METHOD PRIVATE stageEx : BOOL
VAR_IN_OUT
	robot : RobotA21;
	aoiTemplate : AOI_StagingTemplate;
	aoiStaging : AOI_StageWoodBunk;
	stageStep : INT;
END_VAR
VAR_INPUT
	includeTop, includeLeft, includeRight, includeBottom : BOOL;
END_VAR
VAR_OUTPUT
	error : BOOL;
END_VAR
{warning disable C0371}
IF robot.error THEN
	error := TRUE;
	RETURN;
ELSIF robot.reservation <> sectionID AND_THEN NOT robot.reserve(sectionID) THEN
	RETURN;
ELSIF robot.tool <> sectionID AND_THEN NOT robot.changeEOAT(targetTool := sectionID) THEN
	RETURN;
END_IF

CASE stageStep OF
	0: //generate staging template
		IF aoiTemplate.done THEN
			aoiTemplate.execute := FALSE;
			stageStep := 10;
			RETURN;
		END_IF
		
		aoiTemplate.execute := NOT aoiTemplate.busy;
		
		aoiTemplate.includeTop := includeTop;
		aoiTemplate.includeLeft := includeLeft;
		aoiTemplate.includeRight := includeRight;
		aoiTemplate.includeBottom := includeBottom;
		
	10: //stage tables
		IF aoiStaging.slot > 10 THEN
			aoiStaging.execute := FALSE;			
			stageStep := COMPLETE;
			RETURN;
		END_IF
		
		aoiStaging.execute := NOT aoiStaging.busy; //execute if aoiStaging is ready
		
		aoiStaging.slot := MAX(1, aoiStaging.slot); //if 0, sets to 1
		aoiStaging.slot := MIN(aoiStaging.slot, 999); //prevents overflow 
		
		IF aoiStaging.donePulse THEN
			aoiStaging.slot := aoiStaging.slot + 1;
		END_IF
	
	COMPLETE:
		aoiTemplate.clearTemplate();
		aoiTemplate.execute := FALSE;
		aoiStaging.execute := FALSE;
		aoiStaging.reset();
		
		robot.release(sectionID);
		
		aoiStaging.slot := 0;
		
		stageEx := TRUE;
		//stageStep := 0;
END_CASE

error := aoiStaging.error;
END_METHOD

METHOD PROTECTED usesProcess : BOOL
VAR
	i : INT;
END_VAR
FOR i:=0 TO GVL.maxPairs BY 1 DO
	IF PositionIsValid(materialsArr[i]) THEN
		usesProcess := TRUE;
		RETURN;
	END_IF
END_FOR
END_METHOD

METHOD PROTECTED validateInsertion : BOOL
VAR_INPUT
	checkTop : BOOL;
	checkLeft : BOOL;
	checkRight : BOOL;
	checkBottom : BOOL;
END_VAR
validateInsertion := 
	(NOT checkTop OR_ELSE SuctionQuality(suctions:= suctionTop)) AND
	(NOT checkLeft OR_ELSE SuctionQuality(suctions:= suctionLeft)) AND
	(NOT checkRight OR_ELSE SuctionQuality(suctions:= suctionRight)) AND
	(NOT checkBottom OR_ELSE SuctionQuality(suctions:= suctionBottom));

(*
validateSuctionQuality := 
	(
		NOT checkTop OR_ELSE InsertionQuality(
			suctions:= suctionTop, 
			insertionMaterial:= loadedMaterials[Surface.TOP], 
			recipeMaterial:= materialsArr[iPair].top)
	) AND
	(
		NOT checkLeft OR_ELSE InsertionQuality(
			suctions:= suctionLeft, 
			insertionMaterial:= loadedMaterials[Surface.LEFT], 
			recipeMaterial:= materialsArr[iPair].left)
	) AND
	(
		NOT checkRight OR_ELSE InsertionQuality(
			suctions:= suctionRight, 
			insertionMaterial:= loadedMaterials[Surface.RIGHT], 
			recipeMaterial:= materialsArr[iPair].right)
	) AND
	(
		NOT checkBottom OR_ELSE InsertionQuality(
			suctions:= suctionBottom, 
			insertionMaterial:= loadedMaterials[Surface.BOTTOM], 
			recipeMaterial:= materialsArr[iPair].bottom)
	);
*)
END_METHOD

END_FUNCTION_BLOCK

// ---- Sections/Abstract/SectionEx.TcPOU
FUNCTION_BLOCK ABSTRACT SectionEx
VAR_INPUT
	enable : BOOL;
	sectionID : SectionEnum;
	
	firstConveyor : INT;
	lastConveyor : INT;
END_VAR
VAR_IN_OUT
	bundlesQueue : ARRAY[*] OF Bundle;
	bundlesBypass : ARRAY[*] OF BOOL; //if true, then bypass current bundle
END_VAR
VAR_OUTPUT
	bundleOut : Bundle; //assigned if there is a bundle to target
	bypass : BOOL; //assigned once the bundle head passes the section (status >= ACTIVE)
END_VAR
VAR_OUTPUT //PackML states + controls
	pmlModeString : STRING;
	pmlStateString : STRING;
	
	stop : BOOL;
	execute : BOOL;
	hold : BOOL;
	reset : BOOL;
	
	ready : BOOL;
	busy : BOOL;
	done : BOOL;
	error : BOOL;
	backlog : BOOL;
	
	iBundle : INT(0..GVL.maxQueue);
	iPair : INT(0..GVL.maxPairs);
END_VAR
VAR
	pmlState : E_PMLState;
	pmlCommand : E_PMLCommand;
	pmlStateMachine : PML_StateMachine;
	
	pmlModeRequest : E_PMLCustomUnitMode := ePMLCustomUnitMode_Production;
	pmlMode : E_PMLCustomUnitMode;
	pmlModeManager : PML_UnitModeManager;
END_VAR
VAR
	currentBundle : REFERENCE TO Bundle;
	currentBypass : REFERENCE TO BOOL;
	
	loaded : BOOL;
	loadedMaterials : ARRAY[Surface.TOP..Surface.BOTTOM_RIGHT] OF STRING;
	
	entryRefPos : (*REFERENCE TO*) REAL;
	exitRefPos : (*REFERENCE TO*) REAL;
	
	requestedConveyorMode : ConveyorMode;
	
	nextSection : POINTER TO SectionEx;
	prevSection : POINTER TO SectionEx;
	
	occupied : BOOL; //may need to move this to Hardware GVL since this is a sensor
	
	status : SectionTask; //section status
END_VAR
VAR_STAT CONSTANT
	INCLUSIVE : INT := 0;
	EXCLUSIVE : INT := 1;
	COMPLETE : INT := 1030;
	
	suctionReleaseDelay : TIME := T#1000MS;
END_VAR

currentBundle REF= bundlesQueue[iBundle];
currentBypass REF= bundlesBypass[iBundle];
bypass := currentBypass;

ready := status = 0;
busy := status > 0;
done := done;
error := error;
backlog := iBundle >= GVL.maxQueue;

callLocalModules();
blocks();

pmlStates();

METHOD assignConveyors : BOOL
VAR_INPUT
	conveyorStart : INT;
	conveyorEnd : INT;
END_VAR
firstConveyor := conveyorStart;
lastConveyor := conveyorEnd;

assignConveyors := TRUE;
END_METHOD

METHOD PROTECTED blocks : BOOL
VAR_INPUT
END_VAR
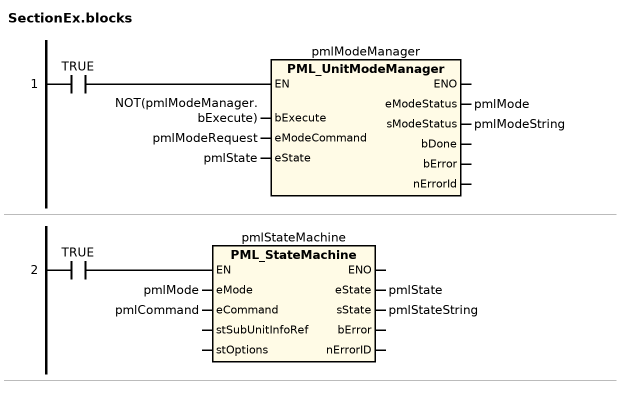
// NETWORK 1
pmlModeManager(
    bExecute := NOT(pmlModeManager.bExecute),
    eModeCommand := pmlModeRequest,
    eState := pmlState,
    eModeStatus => pmlMode,
    sModeStatus => pmlModeString); // PML_UnitModeManager

// NETWORK 2
pmlStateMachine(eMode := pmlMode, eCommand := pmlCommand, eState => pmlState, sState => pmlStateString); // PML_StateMachine
END_METHOD

METHOD PROTECTED ABSTRACT callLocalModules : BOOL
END_METHOD

METHOD connectTo : BOOL
VAR_INPUT
	connectedSection : POINTER TO SectionEx;
END_VAR
nextSection := connectedSection;

IF connectedSection <> 0 THEN
	connectedSection^.prevSection := THIS;
END_IF
END_METHOD

METHOD PROTECTED directionCheckAndSet : BOOL
VAR_INPUT
	conveyorRef : REAL;
	target : REAL;
END_VAR
//returns true conveyorRef is in range of target
IF InRange(conveyorRef - GVL.precisionTolerance, conveyorRef + GVL.precisionTolerance, target, EXCLUSIVE) THEN
	directionCheckAndSet := TRUE;
	
ELSIF conveyorRef > target THEN
	pConveyorMode := ConveyorMode.BACKWARD;
	
ELSIF conveyorRef < target THEN
	pConveyorMode := ConveyorMode.FORWARD;
	
END_IF
END_METHOD

METHOD PROTECTED ABSTRACT discharge : BOOL
VAR_INPUT
END_VAR
(*
unload, unstage, etc
*)
END_METHOD

METHOD PROTECTED ABSTRACT load : BOOL
VAR_INPUT
	pairIndex : INT;
END_VAR
VAR_OUTPUT
	error : BOOL;
END_VAR
(*
loading takes place while the section is NOT active
materials are loaded for the next incoming bundle, not the current bundle - may differ for each section
*)
END_METHOD

METHOD PROTECTED ABSTRACT maintenance : BOOL
VAR_INPUT
END_VAR
END_METHOD

PROPERTY PROTECTED pConveyorMode : ConveyorMode
GET
pConveyorMode := requestedConveyorMode;
END_GET
SET
VAR
	i : DINT;
END_VAR
requestedConveyorMode := pConveyorMode;

FOR i:=firstConveyor TO lastConveyor BY 1 DO
	
	CASE status OF
		SectionTask.ALIGNING, -100:
			//all conveyors requested to same mode
			conveyorsArr[i]^.setRequest(requestedConveyorMode);
			
		SectionTask.ACTIVE, SectionTask.CLEARING:
			//once previous bundle catches up, the conveyor that bundle sits on must be linked to this section
			//a conveyor control module will handle linking
			
			IF conveyorsArr[i]^.IsOccupied THEN //follow this section's request
				conveyorsArr[i]^.setRequest(requestedConveyorMode);
				
			ELSE //catch up succeeding bundle (FOLLOW PREVIOUS SECTION)
				IF prevSection <> 0 THEN
					conveyorsArr[i]^.setRequest( prevSection^.pConveyorMode );
				END_IF
			END_IF
	END_CASE	
	
END_FOR
END_SET
END_PROPERTY

METHOD PROTECTED pmlStates : BOOL
(*
PackML
	state machine for packaging applications - see Tc3_PackML_V2 library on InfoSys
	
	final states - wait for an input or condition and command to new state
	intermediate states - complete a task and call pmlStateMachine.M_StateComplete() to advance to next state
	
the following states currently use the same logic (albeit in different methods), implementation may change later
	ps_Stopping() and ps_Aborting()
	ps_Resetting() and ps_Clearing()
	
STOP - controlled stop **with intent to shutdown or vacate for extended time** induced by operator/HMI - otherwise use HOLD
ABORT - emergency stop due to machine errors


HOLD - minor local issues
SUSPEND - external issues

EXECUTE - major control logic
	different modes may require different tasks
	create methods as required for different modes, then call the correct method in ps_Completing()
	can be commanded to STOP, ABORT, HOLD, or SUSPEND at any point
COMPLETING - process complete, move product out of system and finish transition to COMPLETED

the implementation below can be copied to all POUs that use a PackML state machine
the individual ps_< > methods need to be implemented for the specific application
*)
IF ps_AbortCondition() THEN //abort condition
	pmlCommand := ePMLCommand_Abort;
ELSIF ps_StopCondition() THEN //stop condition
	pmlCommand := ePMLCommand_Stop;
END_IF

CASE pmlState OF
	0 (*ePMLState_Undefined*): //default state on startup
		pmlCommand := ePMLCommand_Stop;
		
	ePMLState_Stopping:
		IF ps_Stopping() THEN
			pmlStateMachine.M_StateComplete();
		END_IF
		
	ePMLState_Stopped:
		IF ps_Stopped() THEN
			pmlCommand := ePMLCommand_Reset;
		END_IF
	
    ePMLState_Resetting:
		IF ps_Resetting() THEN
			pmlStateMachine.M_StateComplete();
		END_IF
		
	ePMLState_Idle:
		IF ps_Idle() THEN
			pmlCommand := ePMLCommand_Start;
		END_IF		
	
	ePMLState_Starting:
		IF ps_Starting() THEN
			pmlStateMachine.M_StateComplete();
		END_IF
	
	ePMLState_Execute: //check the conditions in order of their priority, currently HOLD has the highest priority
		IF ps_HoldCondition() THEN
			pmlCommand := ePMLCommand_Hold;
			
		ELSIF ps_SuspendCondition() THEN
			pmlCommand := ePMLCommand_Suspend;			
		
		ELSIF ps_Execute(error => error) THEN //ps_Execute.error => THIS^.error
			pmlStateMachine.M_StateComplete();
			pmlCommand := ePMLCommand_Complete;
		END_IF
		
	ePMLState_Completing:
		IF ps_Completing() THEN
			pmlStateMachine.M_StateComplete();
		END_IF
	
	ePMLState_Complete:
		IF ps_Complete() THEN
			pmlCommand := ePMLCommand_Reset;
		END_IF
	
	ePMLState_Holding:
		IF ps_Holding() THEN
			pmlStateMachine.M_StateComplete();
		END_IF
	
	ePMLState_Held:
		IF NOT hold THEN
			pmlCommand := ePMLCommand_Unhold;
		END_IF
	
	ePMLState_Unholding:
		IF ps_Unholding() THEN
			pmlStateMachine.M_StateComplete(); //release all pause commands and IO
		END_IF
		
	ePMLState_Suspending: //based on next section conditions
		IF ps_Suspending() THEN
			pmlStateMachine.M_StateComplete();
		END_IF
		
	ePMLState_Suspended: //based on next section conditions
		IF ps_Suspended() THEN
			pmlCommand := ePMLCommand_Unsuspend;
		END_IF
	
	ePMLState_Unsuspending: //based on next section conditions
		IF ps_Unsuspending() THEN
			pmlStateMachine.M_StateComplete();
		END_IF
	
	ePMLState_Aborting:
		IF ps_Aborting() THEN
			pmlStateMachine.M_StateComplete();
		END_IF
	
	ePMLState_Aborted:
		IF ps_Aborted() THEN
			pmlCommand := ePMLCommand_Clear;
		END_IF
	
	ePMLState_Clearing:
		IF ps_Clearing() THEN
			pmlStateMachine.M_StateComplete();
		END_IF
	
END_CASE
END_METHOD

METHOD PROTECTED ABSTRACT process : BOOL
VAR_INPUT
	auto : BOOL;
END_VAR
VAR_OUTPUT
	error : BOOL;
END_VAR
(*
this method is implemented by each section according to their material packaging steps
*)
END_METHOD

METHOD PROTECTED ABSTRACT ps_AbortCondition : BOOL
VAR_INPUT
END_VAR
END_METHOD

METHOD PROTECTED ABSTRACT ps_Aborted : BOOL
VAR_INPUT
END_VAR
END_METHOD

METHOD PROTECTED ABSTRACT ps_Aborting : BOOL
VAR_INPUT
END_VAR
END_METHOD

METHOD PROTECTED ABSTRACT ps_Clearing : BOOL
VAR_INPUT
END_VAR
END_METHOD

METHOD PROTECTED ABSTRACT ps_Complete : BOOL
VAR_INPUT
END_VAR
END_METHOD

METHOD PROTECTED ABSTRACT ps_Completing : BOOL
VAR_INPUT
END_VAR
END_METHOD

METHOD PROTECTED ps_Execute : BOOL
VAR_INPUT
END_VAR
VAR_OUTPUT
	error : BOOL;
END_VAR
CASE pmlMode OF
	0: //invalid mode
	ePMLCustomUnitMode_Production:		ps_Execute := runSectionTasks(auto := TRUE);
	ePMLCustomUnitMode_Maintenance:		maintenance();
	ePMLCustomUnitMode_Manual:			//
	ePMLCustomUnitMode_SemiAuto:		ps_Execute := runSectionTasks(auto := FALSE);
END_CASE
END_METHOD

METHOD PROTECTED ABSTRACT ps_Held : BOOL
VAR_INPUT
END_VAR
END_METHOD

METHOD PROTECTED ABSTRACT ps_HoldCondition : BOOL
VAR_INPUT
END_VAR
END_METHOD

METHOD PROTECTED ABSTRACT ps_Holding : BOOL
VAR_INPUT
END_VAR
END_METHOD

METHOD PROTECTED (*ABSTRACT*) ps_Idle : BOOL
VAR_INPUT
END_VAR
(*
IF BundleIsValid(currentBundle) THEN
	ps_Idle := TRUE;
	done := FALSE;
END_IF
*)

ps_Idle := TRUE; (*start section input*)
END_METHOD

METHOD PROTECTED ABSTRACT ps_Resetting : BOOL
VAR_INPUT
END_VAR
END_METHOD

METHOD PROTECTED ABSTRACT ps_Starting : BOOL
VAR_INPUT
END_VAR
END_METHOD

METHOD PROTECTED ABSTRACT ps_StopCondition : BOOL
VAR_INPUT
END_VAR
END_METHOD

METHOD PROTECTED ABSTRACT ps_Stopped : BOOL
VAR_INPUT
END_VAR
END_METHOD

METHOD PROTECTED ABSTRACT ps_Stopping : BOOL
VAR_INPUT
END_VAR
END_METHOD

METHOD PROTECTED ABSTRACT ps_SuspendCondition : BOOL
VAR_INPUT
END_VAR
END_METHOD

METHOD PROTECTED ABSTRACT ps_Suspended : BOOL
VAR_INPUT
END_VAR
END_METHOD

METHOD PROTECTED ABSTRACT ps_Suspending : BOOL
VAR_INPUT
END_VAR
END_METHOD

METHOD PROTECTED ABSTRACT ps_Unholding : BOOL
VAR_INPUT
END_VAR
END_METHOD

METHOD PROTECTED ABSTRACT ps_Unsuspending : BOOL
VAR_INPUT
END_VAR
END_METHOD

PROPERTY PROTECTED pStatus : SectionTask
GET
pStatus := status;
END_GET
SET
status := pStatus;
END_SET
END_PROPERTY

METHOD PROTECTED FINAL runSectionTasks : BOOL
VAR_INPUT
	auto : BOOL;
END_VAR
VAR
	error : BOOL;
END_VAR
CASE status OF
	SectionTask.IDLE:
		IF BundleIsValid(currentBundle) THEN			
			status := SectionTask.ALIGNING;
			done := FALSE;
		END_IF
	
	SectionTask.ALIGNING:		
		pConveyorMode := ConveyorMode.FORWARD;
		
		IF 
			occupied AND
			nextSection <> 0 AND
			nextSection^.pConveyorMode = ConveyorMode.BACKWARD
		THEN //section occupied by next section backing up into this section
			status := -100;
			
		ELSIF occupied THEN //section occupied by correct bundle
			//stop and zero the conveyors
			IF NOT auto OR_ELSE execute THEN
				status := SectionTask.ACTIVE;
			END_IF
		END_IF
		
	SectionTask.ACTIVE:
		bundleOut := currentBundle;
		
		IF NOT enable THEN
			iPair := 0;
			status := SectionTask.CLEARING;
			
		ELSIF NOT usesProcess() THEN //bundle does not use this section's processes
			iPair := 0;
			status := SectionTask.CLEARING;
		
		ELSIF currentBypass (*AND_THEN discharge()*) THEN //bundle failed in previous section, discharge this section's materials
			IF discharge() THEN
				iPair := 0;
				status := SectionTask.CLEARING;
			END_IF
			
		ELSIF process(auto := auto, error => error) THEN //bundle recipe completed normally
			IF NOT auto OR_ELSE execute THEN
				iPair := 0;
				status := SectionTask.CLEARING;
			END_IF			
		END_IF
		
	SectionTask.CLEARING:
		bundleOut := currentBundle;
		pConveyorMode := ConveyorMode.FORWARD;
		
		IF exitRefPos >= currentBundle.length AND NOT occupied THEN //rear of bundle has cleared the area
			status := SectionTask.COMPLETE;
		END_IF
		
	SectionTask.COMPLETE:	
		iBundle := iBundle + 1;
		//bundleOut := GVL.nullBundle;
		MEMSET(ADR(bundleOut), 0, SIZEOF(bundleOut));
		
		status := SectionTask.IDLE;
		
		runSectionTasks := TRUE;
		
	-100: //previously completed bundle reversed into this section		
		pConveyorMode := ConveyorMode.FORWARD;
		
		IF NOT occupied THEN
			status := SectionTask.ALIGNING;
		END_IF
		
END_CASE
END_METHOD

METHOD shiftIterator : BOOL
VAR
	i : INT;
END_VAR
//2023-10-24 - array of pointers replaced with iterator for MAIN's queue passed by pointer
iBundle := iBundle - 1;
END_METHOD

METHOD PROTECTED ABSTRACT usesProcess : BOOL
(*
this method determines if a bundle uses materials that this section provides
if a bundle does not use this section's process, then it can be skipped
*)
END_METHOD

END_FUNCTION_BLOCK

// ---- Sections/A21b - Wood Bunk/AOIs/AOI_StagingTemplate.TcPOU
FUNCTION_BLOCK AOI_StagingTemplate
VAR_INPUT
	execute : BOOL;
END_VAR
VAR_IN_OUT
	materialsArr : ARRAY[*] OF PositionMaterials; //[0..GVL.maxPairs]
	table : StagingTable;
END_VAR
VAR_INPUT
	includeTop, includeLeft, includeRight, includeBottom : BOOL; 
END_VAR
VAR_OUTPUT
	busy : BOOL;
	done : BOOL;
END_VAR
VAR
	trigger : R_TRIG;
	run : BOOL;
	step : (IDLE, GENERATE, COMPLETE);
	i : INT;
END_VAR
VAR	
	stagingArray : ARRAY[0..(GVL.maxPairs+1)*2] OF STRING;
	
	template : StagingTable;
	templateSlots AT %M* : ARRAY[1..10] OF MaterialSlot;
END_VAR

{warning disable C0371}

template(slots:= templateSlots);

trigger(CLK:= execute, Q=> run);

CASE step OF
	IDLE:
		IF run THEN
			step := GENERATE;
			done := FALSE;
		END_IF
		
	GENERATE:
		//strings contain garbage chars after a null byte, they must be manually cleaned before checking if they are byte-empty
		CleanStringsArray(arr := stagingArray);
		IF DataIsEmtpy(arr := ADR(stagingArray), arrSize := SIZEOF(stagingArray)) THEN //if staging array is empty, fill the array
			createStagingArray(
				includeTop:= includeTop, 
				includeLeft:= includeLeft, 
				includeRight:= includeRight, 
				includeBottom:= includeBottom);
		END_IF
		
		//copy over the real slots before autofilling, otherwise the template may fill occupied slots
		table.copyFrom(src := table);
		
		(*
		iterate through all pairs and autofill the template
		replace succesfully autofilled materials with empty string
		if staging needs to be performed a 2nd time, autofilling empty strings is always unsuccessful
		*)
		FOR i:=0 TO (GVL.maxPairs+1)*2 BY 1 DO
			IF template.autofill(material := stagingArray[i]) THEN
				stagingArray[i] := '';
			END_IF
		END_FOR
		
		step := COMPLETE;
	
	COMPLETE:
		done := TRUE;
		
		step := IDLE;
		
END_CASE

busy := run OR step > 0;

METHOD PRIVATE addToStagingArray : BOOL
VAR_INPUT
	material : STRING;
END_VAR
VAR
	remainingMaterial : STRING;
	splitMaterial : STRING;
END_VAR
remainingMaterial := material;
WHILE FIND(remainingMaterial, '_') > 0 DO
	splitCombinedMaterials(remainingMaterial, splitMaterial);
	IF splitMaterial <> '' THEN
		AddToStringArray(arr := stagingArray, newString := splitMaterial, numElements => , nextIndex => );
	END_IF
END_WHILE

IF remainingMaterial <> '' THEN
	AddToStringArray(arr := stagingArray, newString := remainingMaterial, numElements => , nextIndex => );
END_IF

addToStagingArray := TRUE;
END_METHOD

METHOD clearArray : BOOL
VAR_INPUT
END_VAR
MEMSET(ADR(stagingArray), 0, SIZEOF(stagingArray));
END_METHOD

METHOD clearTemplate : BOOL
VAR_INPUT
END_VAR
template.clear();
END_METHOD

METHOD PRIVATE createStagingArray : BOOL
VAR_INPUT
	includeTop : BOOL;
	includeLeft : BOOL;
	includeRight : BOOL;
	includeBottom : BOOL;
END_VAR
VAR
	remainingMaterial : STRING;
	splitMaterial : STRING;
	
	i : INT;
END_VAR
FOR i:=0 TO GVL.maxPairs BY 1 DO
	IF includeTop THEN
		addToStagingArray(material := materialsArr[i].top);
	END_IF
	
	IF includeLeft THEN
		addToStagingArray(material := materialsArr[i].left);
	END_IF
	
	IF includeRight THEN
		addToStagingArray(material := materialsArr[i].right);
	END_IF
	
	IF includeBottom THEN
		addToStagingArray(material := materialsArr[i].bottom);
	END_IF
END_FOR
END_METHOD

METHOD getSlot : STRING
VAR_INPUT
	i : INT;
END_VAR
VAR_OUTPUT
	error : BOOL;
END_VAR
getSlot := template.getSlot(i := i, error => error);
END_METHOD

METHOD reset : BOOL
VAR_INPUT
END_VAR
VAR
	temp : AOI_StagingTemplate;
END_VAR
//(*
busy := FALSE;
done := FALSE;
step := 0;

clearArray();
clearTemplate();
//*)
//THIS^ := temp;
END_METHOD

METHOD PRIVATE splitCombinedMaterials : BOOL
VAR_IN_OUT
	materialID : STRING;
	splitMaterial : STRING;
END_VAR
VAR
	i : INT;
END_VAR
FindAndSplitChar(
	sSeparatorChar:= '_', 
	pSrcString:= ADR(materialID), 
	
	pLeftString:= ADR(splitMaterial), 
	nLeftSize:= SIZEOF(splitMaterial), 
	
	pRightString:= ADR(materialID), 
	nRightSize:= SIZEOF(materialID), 
	
	bSearchFromRight:= FALSE);
END_METHOD

END_FUNCTION_BLOCK

// ---- Sections/A21b - Wood Bunk/AOIs/AOI_StageWoodBunk.TcPOU
FUNCTION_BLOCK AOI_StageWoodBunk
VAR_INPUT
	execute : BOOL;
END_VAR
VAR_IN_OUT CONSTANT
	sectionID : SectionEnum;
END_VAR
VAR_IN_OUT
	robot : RobotA21;
	table : StagingTable;
	magazine : SkidMagazine;
END_VAR
VAR_INPUT
	slot : INT;
	material : STRING;
END_VAR
VAR_OUTPUT
	busy : BOOL;
	done : BOOL; //this done signal stays on until next execution
	error : BOOL;
	
	recovery : BOOL;
	failCounter : INT;
	
	donePulse : BOOL; //this done signal only stays on for 1 cycle after completion
END_VAR
VAR
	run : BOOL;
	trigger : R_TRIG;	
	doneTrigger : R_TRIG;
	
	column : INT;
	step : (IDLE, PREP_ROBOT, GET_FROM_MAGAZINE, PLACE_ON_TABLE, COMPLETE);
END_VAR
VAR CONSTANT
	suctionDistance : INT := 10;
END_VAR

{warning disable C0371}
{warning disable C0195}
(*
IF error THEN
	step := IDLE;
END_IF
*)
trigger(CLK:= execute, Q=> );
doneTrigger(CLK:= done, Q=> donePulse);

busy := trigger.Q OR step > 0;

IF step > IDLE AND_THEN NOT preExecution() THEN //conditions to track before execution
	RETURN;
END_IF

//follow the template as is
CASE step OF
	IDLE:
		IF trigger.Q THEN //reset outputs
			done := FALSE;
			error := FALSE;
			recovery := FALSE;
			
			step := PREP_ROBOT;
		END_IF
		
	PREP_ROBOT:
		robot.clearCommand();
		IF robot.Ready THEN
			step := GET_FROM_MAGAZINE;
		END_IF
	
	GET_FROM_MAGAZINE: //grab from magazine
		IF NOT magazine.findSlot(material := material, index => column) THEN
			error := TRUE;
			RETURN;
		END_IF
		
		IF robot.eoatDistance < suctionDistance THEN //robot is grabbing material
			robot.HoldMaterial := magazine.getSlot(i := column);
		END_IF
		
		IF robot.Done THEN
			step := COMPLETE;
			RETURN;
		END_IF
		
		robot.setGroup(group := 1, value := A21.STAGE_BUNK);
		robot.setGroup(group := 2, value := column);
		robot.setGroup(group := 3, value := slot);

	COMPLETE: //check here if staging is successful or needs to be repeated
		robot.clearCommand();
		
		IF table.isOccupied(slot) THEN
			table.place(i := slot, materialID := robot.HoldMaterial);
			robot.HoldMaterial := '';
			
			failCounter := 0;
			done := TRUE;
		ELSE
			failCounter := failCounter + 1;
		END_IF
		
		step := 0;
		
END_CASE

METHOD PRIVATE preExecution : BOOL
VAR_INPUT
END_VAR
{warning disable C0371}

IF slot < 1 THEN //out of bounds for staging table
	error := TRUE;
	RETURN;
ELSIF table.isFull() OR slot > 10 OR material = '' OR table.getSlot(i := slot, error => ) = material THEN
	done := TRUE;
	RETURN;
END_IF

IF //robot must be ready before execution
	robot.error OR 
	robot.reservation <> sectionID OR 
	robot.tool <> sectionID
THEN
	error := TRUE;
	RETURN;
END_IF

preExecution := TRUE;
END_METHOD

METHOD reset : BOOL
VAR_INPUT
END_VAR
VAR
	temp : AOI_StageWoodBunk;
END_VAR
//(*
done := FALSE;
error := FALSE;
recovery := FALSE;
slot := 0;
step := 0;

failCounter := 0;
//*)
//THIS^ := temp;
END_METHOD

END_FUNCTION_BLOCK

// ---- Sections/A21b - Wood Bunk/AOIs/AOI_LoadWoodBunk.TcPOU
FUNCTION_BLOCK AOI_LoadWoodBunk
VAR_INPUT
	execute : BOOL;
END_VAR
VAR_IN_OUT CONSTANT
	sectionID : SectionEnum;
END_VAR
VAR_IN_OUT
	robot : RobotA21;
	table : StagingTable;
	suctions : ARRAY[*] OF SuctionPad;
	//if assigned using . operator instead of (), this becomes a pointer - use numPads isntead of UPPER_BOUND/LOWER_BOUND
	loadedMaterials : ARRAY[*] OF STRING;
END_VAR
VAR_INPUT
	surfaceID : Surface;
	material : STRING;	
	numPads : DINT;
END_VAR
VAR_OUTPUT
	busy : BOOL;
	done : BOOL;
	error : BOOL;
	
	recovery : BOOL;
	failCounter : INT;
	
	donePulse : BOOL;
END_VAR
VAR
	run : BOOL;
	trigger : R_TRIG;
	doneTrigger : R_TRIG;
	
	slot : INT;
	
	suctionTimer : TON;
	step : (IDLE, PREP_ROBOT, GET_FROM_TABLE, LOAD_TO_INSERTION, COMPLETE, RECOVERY_IDLE, RECOVERY_REMOVE, RECOVERY_STAGE);
END_VAR
VAR
	i : DINT;
	test : BOOL;
END_VAR
VAR CONSTANT
	suctionDelay : TIME := T#2S;
	suctionDistance : INT := 10;
END_VAR

{warning disable C0371}

trigger(CLK:= execute, Q=> );
doneTrigger(CLK:= done, Q=> donePulse);
busy := trigger.Q OR step > 0;

IF step > IDLE AND_THEN NOT preExecution() THEN //conditions to track before execution
	RETURN;
END_IF

(*
if required bunk was not found on table - restage entire table
if bunk was not loaded correctly - remove bunk, then restage entire table
*)

CASE step OF
	IDLE:
		IF trigger.Q THEN //reset outputs
			done := FALSE;
			error := FALSE;
			recovery := FALSE;
			
			step := PREP_ROBOT;
		END_IF
		
	PREP_ROBOT:
		robot.clearCommand();
		IF robot.Ready THEN
			step := GET_FROM_TABLE;
			slot := 0;
		END_IF
		
	GET_FROM_TABLE:		
		IF slot < 1 AND_THEN NOT table.findSlot(material := material, index => slot) THEN
			step := RECOVERY_STAGE;
			RETURN;
		END_IF
		
		IF NOT table.isOccupied(i := slot) AND table.getSlot(i := slot) <> '' THEN //move from table to robot gripper
			robot.HoldMaterial := table.getSlot(i := slot);
			table.remove(i := slot, material => );
		END_IF
		
		IF robot.Done THEN
			step := COMPLETE;
			RETURN;
		ELSIF robot.materialAtHoldingPosition >= 1 AND robot.materialAtHoldingPosition <= 8 THEN
			step := LOAD_TO_INSERTION;
			RETURN;
		END_IF
		
		CASE surfaceID OF
			Surface.TOP: 					robot.setGroup(group := 1, value := A21.LOAD_BUNK_TOP); 
			Surface.LEFT, Surface.RIGHT: 	robot.setGroup(group := 1, value := A21.LOAD_BUNK_SIDE);
			Surface.BOTTOM: 				robot.setGroup(group := 1, value := A21.LOAD_BUNK_BOTTOM);
		END_CASE
		robot.setGroup(group := 2, value := slot); 
			
	LOAD_TO_INSERTION:
		IF robot.materialAtHoldingPosition > 0 AND robot.HoldMaterial <> '' THEN //move from gripper to insertion
			IF loadedMaterials[surfaceID] = '' THEN //transfer to insertion as is
				loadedMaterials[surfaceID] := robot.HoldMaterial;
			ELSE //join with existing material using underscore _
				loadedMaterials[surfaceID] := JoinStrings(loadedMaterials[surfaceID], robot.HoldMaterial, '_');
			END_IF
			robot.HoldMaterial := '';
		END_IF
		
		CASE surfaceID OF
			Surface.TOP, Surface.BOTTOM:	SetSuctionsPtrArr(suctions := suctions, numPads := numPads, state := TRUE);
			Surface.LEFT, Surface.RIGHT:	SetSuctionsPtrArr(suctions := suctions, numPads := numPads, state := TRUE);
		END_CASE
		
		IF robot.Done THEN
			suctionTimer.IN := FALSE;
			step := COMPLETE;
			RETURN;
		END_IF
		
		suctionTimer(IN:= , PT:= suctionDelay, Q=> , ET=> );
		suctionTimer.IN := TRUE;
		
		IF suctionTimer.Q THEN
			robot.setGroup(group := 9, value := robot.materialAtHoldingPosition);
		END_IF
	
	COMPLETE:
		robot.clearCommand();
		
		//check insertion quality
		IF InsertionQuality(suctions := suctions, insertionMaterial := loadedMaterials[surfaceID], recipeMaterial := material) THEN
			done := TRUE;
			slot := 0;
			step := 0;
		ELSE //recovery - restage table
			failCounter := failCounter + 1;
			step := RECOVERY_IDLE;
		END_IF
		
	//---------RECOVERY-----------------------------------------
	RECOVERY_IDLE:
		robot.clearCommand();
		IF robot.Ready THEN
			step := RECOVERY_REMOVE;
		END_IF
		
	RECOVERY_REMOVE:
		IF robot.Done THEN
			step := RECOVERY_STAGE;
			RETURN;
		END_IF
		
		CASE surfaceID OF
			Surface.TOP:					robot.setGroup(group := 1, value := A21.REMOVE_BUNK_TOP);
			Surface.LEFT, Surface.RIGHT:	robot.setGroup(group := 1, value := A21.REMOVE_BUNK_SIDE);
			Surface.BOTTOM:					robot.setGroup(group := 1, value := A21.REMOVE_BUNK_BOTTOM);
		END_CASE
	
	RECOVERY_STAGE:	
		recovery := TRUE;
		error := TRUE;
		
END_CASE

METHOD PRIVATE preExecution : BOOL
VAR_INPUT
END_VAR
{warning disable C0371}
IF material = '' THEN
	done := TRUE;
	RETURN;
END_IF

IF //robot must be ready before execution
	robot.error OR 
	robot.reservation <> sectionID OR 
	robot.tool <> sectionID
THEN
	error := TRUE;
	RETURN;
END_IF

preExecution := TRUE;
END_METHOD

METHOD reset : BOOL
VAR_INPUT
END_VAR
VAR
	temp : AOI_LoadWoodBunk;
END_VAR
//(*
done := FALSE;
error := FALSE;
recovery := FALSE;
slot := 0;
step := 0;

failCounter := 0;
//*)
//THIS^ := temp;
END_METHOD

END_FUNCTION_BLOCK

// ---- Sections/A21a - Chipboard/AOIs/AOI_LoadChipboard.TcPOU
FUNCTION_BLOCK AOI_LoadChipboard
VAR_IN_OUT CONSTANT
	sectionID : SectionEnum;
END_VAR
VAR_INPUT
	execute : BOOL;
END_VAR
VAR_IN_OUT
	robot : RobotA21;
	storage : SkidMagazine;
	loadedMaterials : ARRAY[*] OF STRING;
END_VAR
VAR_INPUT
	surfaceID : Surface;
	material : STRING;
END_VAR
VAR_OUTPUT
	busy : BOOL;
	done : BOOL;
	error : BOOL;
	
	recovery : BOOL;
	failCounter : INT;
	
	donePulse : BOOL;
END_VAR
VAR
	run : BOOL;
	trigger : R_TRIG;
	doneTrigger : R_TRIG;
	
	step : (IDLE, PREP_ROBOT, RETRACT_CONVEYORS, GET_FROM_SKID, LOAD_TO_BUNDLE, COMPLETE);
	column : INT;
END_VAR
VAR CONSTANT
	suctionDistance : INT := 10;
END_VAR

{warning disable C0371}

trigger(CLK:= execute, Q=> );
doneTrigger(CLK:= done, Q=> donePulse);
busy := trigger.Q OR step > 0;

IF step > IDLE AND_THEN NOT preExecution() THEN //conditions to track before execution
	RETURN;
END_IF

trigger(CLK:= execute, Q=> run);

CASE step OF
	IDLE:
		IF trigger.Q THEN //reset outputs
			done := FALSE;
			error := FALSE;
			recovery := FALSE;
			
			step := PREP_ROBOT;
		END_IF
	
	PREP_ROBOT:
		robot.clearCommand();
		IF robot.Ready THEN
			step := RETRACT_CONVEYORS;
		END_IF
	
	RETRACT_CONVEYORS:
		IF surfaceID = Surface.BOTTOM (*AND_THEN conveyors not retracted*) THEN
			//retract conveyors
			RETURN;
		END_IF
		step := GET_FROM_SKID;
		
	GET_FROM_SKID: //grab from chipboard skid
		IF NOT storage.findSlot(material := material, index => column) THEN
			error := TRUE;
			RETURN;
		(*
		ELSIF surfaceID = Surface.BOTTOM (*AND_THEN (*conveyor not lowered*)*) THEN
			//lower conveyor
			RETURN;
		*)
		END_IF
		
		IF robot.eoatDistance < suctionDistance THEN
			robot.HoldMaterial := storage.getSlot(i := column);
		END_IF
		
		IF robot.Done THEN
			step := COMPLETE;
			RETURN;
		ELSIF robot.materialAtHoldingPosition.4 OR robot.materialAtHoldingPosition.5 THEN //bits 4 and 5 = chipboard in position
			step := LOAD_TO_BUNDLE;
			RETURN;
		END_IF
		CASE surfaceID OF
			Surface.TOP:		robot.setGroup(group := 1, value := A21.PLACE_CHIPBOARD_TOP);
			Surface.BOTTOM:		robot.setGroup(group := 1, value := A21.PLACE_CHIPBOARD_BOTTOM);
		END_CASE
		robot.setGroup(group := 2, value := column);
		
	LOAD_TO_BUNDLE: //place to bundle
		IF robot.Done THEN
			step := COMPLETE;
			RETURN;
		END_IF
		
		IF robot.HoldMaterial <> '' THEN
			loadedMaterials[surfaceID] := robot.HoldMaterial;
			robot.HoldMaterial := '';
		END_IF
		
	COMPLETE:
		IF loadedMaterials[surfaceID] = material THEN
			done := TRUE;
			failCounter := 0;
		ELSE
			error := TRUE;
			failCounter := failCounter + 1;
		END_IF
		step := 0;
END_CASE

busy := run OR step > 0;

METHOD PRIVATE preExecution : BOOL
VAR_INPUT
END_VAR
{warning disable C0371}
IF material = '' THEN
	done := TRUE;
	RETURN;
END_IF

IF //robot must be ready before execution
	robot.error OR 
	robot.reservation <> sectionID OR 
	robot.tool <> sectionID
THEN
	error := TRUE;
	RETURN;
END_IF

preExecution := TRUE;
END_METHOD

METHOD reset : BOOL
VAR_INPUT
END_VAR
VAR
	temp : AOI_LoadChipboard;
END_VAR
//(*
done := FALSE;
error := FALSE;
recovery := FALSE;
column := 0;
step := 0;

failCounter := 0;
//*)
//THIS^ := temp;
END_METHOD

END_FUNCTION_BLOCK

// ---- Sections/A21a - Chipboard/ChipboardEx.TcPOU
FUNCTION_BLOCK ChipboardEx EXTENDS SectionEx
VAR_IN_OUT //references to required hardware
	robotLeft, robotRight : RobotA21;
	toolStorageLeft, toolStorageRight : A21ToolStorage;
	
	skidLeft, skidRight : SkidMagazine;
END_VAR
VAR	
	step : (IDLE, RETRACT_CONVEYOR, LOAD_CIP, EXTEND_CONVEYOR, COMPLETE := 1050);
	
	loadSet : INT;
END_VAR
VAR //bundle data
	materialsArr : (*REFERENCE TO*) ARRAY[0..GVL.maxPairs] OF PositionMaterials;
END_VAR
VAR
	aoiLoadLeft, aoiLoadRight : AOI_LoadChipboard;
	
	pushSmallConveyorPos : REAL;
	pushLargeConveyorPos : REAL;
END_VAR

{warning disable C0371}
callLocalModules(); //call local modules

blocks(); //call AOIs and large library FBs

runPML(); //run PackML state machine

ACTION blocks:
aoiLoadRight(
	sectionID:= sectionID, 
	execute:= ,
	robot:= robotRight, 
	storage:= skidRight,
	loadedMaterials:= loadedMaterials,
	surfaceID:= , 
	material:= , 
	loadedMaterials=> , 
	done=> , 
	error=> );
	
aoiLoadRight(
	sectionID:= sectionID, 
	execute:= , 
	robot:= robotRight, 
	storage:= skidRight,
	loadedMaterials:= loadedMaterials, 
	surfaceID:= , 
	material:= , 
	busy=> , 
	done=> , 
	error=> , 
	recovery=> , 
	failCounter=> );
END_ACTION

METHOD PRIVATE callLocalModules : BOOL
END_METHOD

METHOD PROTECTED load : BOOL
VAR_INPUT
	pairIndex : INT;
END_VAR
VAR_OUTPUT
	error : BOOL;
END_VAR
VAR
	pair : REFERENCE TO PositionMaterials REF= materialsArr[pairIndex];
END_VAR
{warning disable C0371}
IF robotLeft.error AND robotLeft.error THEN
	error := TRUE;
	RETURN;

ELSIF
	( robotLeft.reservation <> sectionID AND_THEN robotLeft.reserve(sectionID) ) OR
	( robotRight.reservation <> sectionID AND_THEN robotRight.reserve(sectionID) ) THEN
	RETURN;
	
ELSIF //wrong tool and not finished changing tool
	(robotLeft.tool <> sectionID AND_THEN NOT robotLeft.changeEOAT(targetTool := sectionID)) OR
	(robotRight.tool <> sectionID AND_THEN NOT robotRight.changeEOAT(targetTool := sectionID))
THEN
	RETURN;
END_IF
//robots ok

CASE loadSet OF
	0: //left robot -> top, right robot -> bottom
		IF aoiLoadLeft.done AND aoiLoadRight.done THEN
			aoiLoadLeft.execute := aoiLoadRight.execute := FALSE;
			loadSet := 10;
			RETURN;
		END_IF
		
		aoiLoadLeft.surfaceID := Surface.TOP;
		aoiLoadLeft.material := pair.left;
		
		aoiLoadRight.surfaceID := Surface.BOTTOM;
		aoiLoadRight.material := pair.right;
		
		aoiLoadLeft.execute := NOT aoiLoadLeft.recovery;
		aoiLoadRight.execute := NOT aoiLoadRight.recovery;
		
	10: //recovery		
		IF robotRight.error THEN //left ok, right error
			
			IF aoiLoadLeft.done THEN
				aoiLoadLeft.execute := FALSE;
				loadSet := COMPLETE;
				RETURN;
			END_IF
			
			aoiLoadLeft.surfaceID := Surface.BOTTOM;
			aoiLoadLeft.material := pair.bottom;
			aoiLoadLeft.execute := NOT aoiLoadLeft.recovery;
			
		ELSIF robotLeft.error THEN //left error, right ok
			
			IF aoiLoadRight.done THEN
				aoiLoadRight.execute := FALSE;
				loadSet := COMPLETE;
				RETURN;
			END_IF
			
			aoiLoadRight.surfaceID := Surface.TOP;
			aoiLoadRight.material := pair.top;
			aoiLoadRight.execute := NOT aoiLoadRight.recovery;
			
		END_IF
		
	COMPLETE:
		loadSet := 0;
		
		robotLeft.release(sectionID);
		robotRight.release(sectionID);
		
		load := TRUE;
END_CASE
END_METHOD

METHOD PRIVATE loadingSequence : BOOL
VAR_IN_OUT
	robot : RobotA21;
	storage : SkidMagazine;
	loadStep : INT;
END_VAR
VAR_INPUT
	surfaceID : Surface;
	material : STRING;
END_VAR
VAR_OUTPUT
	fail : BOOL;
END_VAR
VAR
	slot : INT;
END_VAR
VAR CONSTANT
	suctionDistance : INT := 10;
END_VAR
{warning disable C0371}
IF material = '' THEN
	loadingSequence := TRUE;
	RETURN;
END_IF

CASE loadStep OF
	0:
		robot.clearCommand();
		IF robot.Ready THEN
			loadStep := 1;
		END_IF
	
	1:
		IF surfaceID = Surface.BOTTOM (*AND_THEN conveyors not retracted*) THEN
			//retract conveyors
			RETURN;
		END_IF
		loadStep := 10;
		
	10: //grab from chipboard skid
		IF NOT storage.findSlot(material := material, index => slot) THEN
			fail := TRUE;
			RETURN;
		(*
		ELSIF surfaceID = Surface.BOTTOM (*AND_THEN (*conveyor not lowered*)*) THEN
			//lower conveyor
			RETURN;
		*)
		END_IF
		
		IF robot.eoatDistance < suctionDistance THEN
			robot.HoldMaterial := storage.getSlot(i := slot);
		END_IF
		
		IF robot.Done THEN
			loadStep := COMPLETE;
			RETURN;
		ELSIF robot.materialAtHoldingPosition.4 OR robot.materialAtHoldingPosition.5 THEN //bits 4 and 5 are chipboard in position
			loadStep := 20;
			RETURN;
		END_IF
		
		robot.setGroup(group := 1, value := A21.PLACE_CHIPBOARD_TOP);
		robot.setGroup(group := 2, value := slot);
		
	20: //place to bundle
		IF robotLeft.Done THEN
			loadStep := COMPLETE;
			RETURN;
		END_IF
		
		IF robot.HoldMaterial <> '' THEN
			loadedMaterials[surfaceID] := robot.HoldMaterial;
			robot.HoldMaterial := '';
		END_IF
		
	COMPLETE:
		IF loadedMaterials[surfaceID] = material THEN
			loadingSequence := TRUE;
		ELSE
			loadStep := 0;
		END_IF
		
END_CASE
END_METHOD

METHOD PRIVATE maintenance : BOOL
VAR_INPUT
END_VAR
{warning disable C0371}
//no specific tasks yet, free run and testing

IF robotLeft.Done THEN
	robotLeft.clearCommand();
END_IF

IF robotRight.Done THEN
	robotRight.clearCommand();
END_IF
END_METHOD

METHOD PROTECTED process : BOOL
VAR_INPUT
	manualMode : BOOL;
END_VAR
VAR_OUTPUT
	error : BOOL;
END_VAR
CASE step OF
	IDLE:
		IF execute THEN
			execute := FALSE;
			step := RETRACT_CONVEYOR;
		END_IF
		
	RETRACT_CONVEYOR:
		(*
		IF demoPair.bottom <> '' (*retract conveyors*) THEN
			IF TRUE (*BLSC 1-3 retracted*) THEN
				done := TRUE;
			END_IF
		ELSE
			done := TRUE;
		END_IF
		
		IF
			(manualStep AND_THEN execute) OR
			(NOT manualStep AND_THEN done)
		THEN
			done := FALSE;
			step := LOAD_MATERIAL;
		END_IF
		*)
		step := LOAD_CIP;
	LOAD_CIP:
		IF NOT done THEN
			done := load(pairIndex:= iPair, error=> error);
		END_IF
		
		IF
			(manualMode AND_THEN execute) OR
			(NOT manualMode AND_THEN done)
		THEN
			done := FALSE;
			execute := FALSE;
			
			step := EXTEND_CONVEYOR;
		END_IF
		
	EXTEND_CONVEYOR:
		(*
		IF FALSE (*conveyors not extended*) THEN
			//extend conveyors
		END_IF
		
		IF
			(manualStep AND_THEN execute) OR
			(FALSE) //conveyors extended
		THEN
			done := FALSE;
			step := COMPLETE;
		END_IF
		*)
		step := COMPLETE;
	COMPLETE:
		//reset everything
		step := IDLE;
		
		process := TRUE;
		
END_CASE
END_METHOD

METHOD PROTECTED ps_Aborting : BOOL
VAR_INPUT
END_VAR
{warning disable C0371}
aoiLoadLeft.reset();
aoiLoadRight.reset();

robotLeft.clearCommand();
robotRight.clearCommand();

//stop conveyors

ps_Aborting :=
	NOT robotLeft.Busy AND
	NOT robotRight.Busy;
END_METHOD

METHOD PROTECTED ps_Clearing : BOOL
VAR_INPUT
END_VAR
{warning disable C0371}
(*reset conveyors*)

ps_Clearing := 
	NOT robotLeft.error AND
	NOT robotRight.error;
END_METHOD

METHOD PROTECTED ps_Execute : BOOL
VAR_INPUT
END_VAR
VAR_OUTPUT
	error : BOOL;
END_VAR
CASE pmlMode OF
	0: //invalid mode
	ePMLProtUnitMode_Production:	ps_Execute := process(manualMode := FALSE, error => error);
	ePMLProtUnitMode_Maintenance:	maintenance();
	ePMLProtUnitMode_Manual:		ps_Execute := process(manualMode := TRUE, error => error);
END_CASE
END_METHOD

METHOD PROTECTED ps_Holding : BOOL
VAR_INPUT
END_VAR
{warning disable C0371}
//set robot to pause

ps_Holding := TRUE;
END_METHOD

METHOD PROTECTED ps_Resetting : BOOL
VAR_INPUT
END_VAR
{warning disable C0371}
(*reset conveyors*)

ps_Resetting := 
	reset AND
	NOT robotLeft.error AND
	NOT robotRight.error;
END_METHOD

METHOD PROTECTED ps_Starting : BOOL
VAR_INPUT
END_VAR
{warning disable C0371}
//extend conveyors

ps_Starting := TRUE; //conveyors extended
END_METHOD

METHOD PROTECTED ps_Stopping : BOOL
VAR_INPUT
END_VAR
{warning disable C0371}
aoiLoadLeft.reset();
aoiLoadRight.reset();

robotLeft.clearCommand();
robotRight.clearCommand();

//stop conveyors

ps_Stopping :=
	NOT robotLeft.Busy AND
	NOT robotRight.Busy;
END_METHOD

ACTION runPML:
(*
PackML
	state machine for packaging applications - see Tc3_PackML_V2 library on InfoSys
	
	final states - wait for an input or condition and command to new state
	intermediate states - complete a task and call pmlStateMachine.M_StateComplete() to advance to next state
	
the following states currently use the same logic (albeit in different methods), implementation may change later
	ps_Stopping() and ps_Aborting()
	ps_Resetting() and ps_Clearing()
	
STOP - controlled stop **with intent to shutdown or vacate for extended time** induced by operator/HMI - otherwise use HOLD
ABORT - emergency stop due to machine errors


HOLD - minor local issues
SUSPEND - external issues

EXECUTE - major control logic
	different modes may require different tasks
	create methods as required for different modes, then call the correct method in ps_Completing()
	can be commanded to STOP, ABORT, HOLD, or SUSPEND at any point
COMPLETING - process complete, move product out of system and finish transition to COMPLETED
*)

IF //abort at machine error
	robotLeft.error OR 
	robotRight.error
	//+conveyor errors
THEN
	pmlCommand := ePMLCommand_Abort;
	
ELSIF stop THEN //stop at command stop
	pmlCommand := ePMLCommand_Stop;

ELSIF FALSE (*A2.4 cannot allow bundles to enter*) THEN //FALSE condition never executes - this is temporary
	pmlCommand := ePMLCommand_Suspend;
END_IF


CASE pmlState OF
	0: (*ePMLState_Undefined*) //default state on startup
		pmlCommand := ePMLCommand_Stop;
		
	ePMLState_Stopping:
		IF ps_Stopping() THEN
			pmlStateMachine.M_StateComplete();
		END_IF
		
	ePMLState_Stopped:
		pmlCommand := ePMLCommand_Reset;
	
    ePMLState_Resetting:
		IF ps_Resetting() THEN
			reset := FALSE;
			pmlStateMachine.M_StateComplete();
		END_IF
		
	ePMLState_Idle:
		IF execute THEN
			execute := FALSE;
			pmlCommand := ePMLCommand_Start;
		END_IF
	
	ePMLState_Starting:
		IF ps_Starting() THEN
			pmlStateMachine.M_StateComplete();
		END_IF
	
	ePMLState_Execute: 
		IF hold THEN
			pmlCommand := ePMLCommand_Hold;
		END_IF
		IF ps_Execute(error => error) THEN
			pmlStateMachine.M_StateComplete();
			pmlCommand := ePMLCommand_Complete;
		END_IF
		
	ePMLState_Completing:
		pmlStateMachine.M_StateComplete();
	
	ePMLState_Complete:
		pmlCommand := ePMLCommand_Reset;
	
	ePMLState_Holding:
		IF ps_Holding() THEN
			pmlStateMachine.M_StateComplete();
		END_IF
	
	ePMLState_Held:
		IF NOT hold THEN
			pmlCommand := ePMLCommand_Unhold;
		END_IF
	
	ePMLState_Unholding:
		pmlStateMachine.M_StateComplete(); //release all pause commands and IO
	
	ePMLState_Suspended: //based on output section conditions
	ePMLState_Suspending: //based on output section conditions
	ePMLState_Unsuspending: //based on output section conditions
	
	ePMLState_Aborting:
		IF ps_Aborting() THEN
			pmlStateMachine.M_StateComplete();
		END_IF
	
	ePMLState_Aborted:
		pmlCommand := ePMLCommand_Clear;
	
	ePMLState_Clearing:
		IF ps_Clearing() THEN
			pmlStateMachine.M_StateComplete();
		END_IF
	
END_CASE
END_ACTION

END_FUNCTION_BLOCK
